// LS Electric XG5000 project: 2023-08-17 #3
// PLC NewPLC
// module base 0 slot 0: 입력 모듈:XGI-D22A/B (DC 24V 입력, 16점 (전류소스 싱크공용/ 전류소스 입력))
// module base 0 slot 1: 입력 모듈:XGI-D22A/B (DC 24V 입력, 16점 (전류소스 싱크공용/ 전류소스 입력))
// module base 0 slot 2: 출력 모듈:XGQ-RY2A/B (릴레이 출력, 16점 (2A용, Varistor 없음/Varistor 부착))
// module base 0 slot 3: 출력 모듈:XGQ-TR2A/B (트랜지스터 출력, 16점 (0.5A용, 싱크출력/소스출력))

PROGRAM NewProgram (task: 스캔 프로그램)

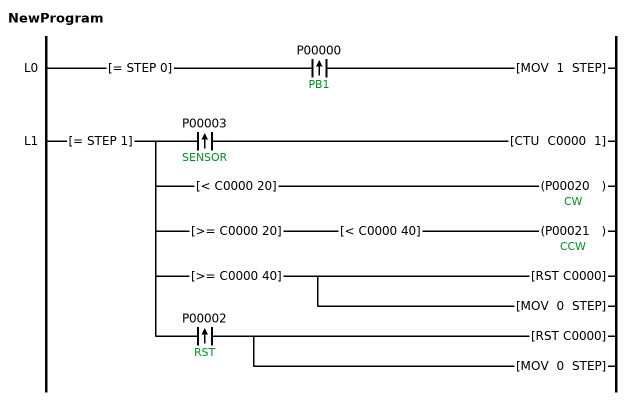
; L0
LOAD=     STEP 0
ANDP      P00000	// PB1
MOV       1 STEP
; L1
LOAD=     STEP 1
MPUSH
ANDP      P00003	// SENSOR
CTU       C0000 1
MLOAD
AND<      C0000 20
OUT       P00020	// CW
MLOAD
AND>=     C0000 20
AND<      C0000 40
OUT       P00021	// CCW
MLOAD
AND>=     C0000 40
RST       C0000
MOV       0 STEP
MPOP
ANDP      P00002	// RST
RST       C0000
MOV       0 STEP

VARIABLES AND COMMENTS (devices not used above)
P00001	BIT	PB2
D00000	WORD	STEP